{attribute 'qualified_only'}
{attribute 'strict'}
{attribute 'to_string'}
TYPE E_EtherCatState :
(
	Unknown,
	Init,
	PreOp,
	BootStrap,
	SafeOp,
	Op,
	Disabled,
	Error
) := Unknown ;
END_TYPE

(* stored: Version 1.1.0.1, ProductVersion 3.1.4024.12
   DUT E_EtherCatState: Id {ebbf2a46-f7a8-47ab-940a-4d7d3ffdf70b} *)
